TYPE SuperimposedActural :
STRUCT
	Done               : BOOL;
    Busy               : BOOL;
    Active             : BOOL;
    CommandAborted     : BOOL;
    Error              : BOOL;
    ErrorID            : UDINT;
	Warning            : BOOL;
    WarningID          : UDINT;
    ActualVelocityDiff : LREAL;
    ActualDistance     : LREAL;
    ActualLength       : LREAL;
    ActualAcceleration : LREAL;
    ActualDeceleration : LREAL;
END_STRUCT
END_TYPE

(* stored: Version 1.1.0.1, ProductVersion 3.1.4024.4
   DUT SuperimposedActural: Id {2f368bb4-bee1-4a4d-aa56-cf537fb40c6c} *)
